// TIA Portal V20 export
DATA_BLOCK "Et200SpMotorstarterInterfaceHmi"   // DB208
// stored: InstanceOfName typeEt200SpMotorstarterInterfaceHmi, InstanceOfType UDT
"typeEt200SpMotorstarterInterfaceHmi"
   // VAR
   //    et200SpMotorstarterReadValue : Bool;
   //    et200SpNumberOfMotorstarters { ExternalWritable := 'False'} : USInt;
   //    et200SpUnitMotorstarter : USInt;
   //    et200SpEMMotorstarter : USInt;
   //    et200SpMotorstarterCurrent : Array[0.."NO_OF_ET200SPMOTORSTARTER"] of Real;
   //    et200SpMotorstarterInputs : Array[0.."NO_OF_ET200SPMOTORSTARTER"] of "LSicar_typeMotorstarterIn";
   //    et200SpMotorstarterOutputs : Array[0.."NO_OF_ET200SPMOTORSTARTER"] of "LSicar_typeMotorstarterOut";
   // END_VAR
BEGIN
END_DATA_BLOCK
